Universal Robots PolyScope program: cognex01.urp

Program cognex01 (installation=default directory=/programs createdIn=5.9.1.1031110 lastSavedIn=5.9.1.1031110 robotSerialNumber=20195501059)
Calibrated DH parameters: a=[0.000146, -0.418764, -0.053981, 0.000058, -0.000023, 0]; d=[0.162545, 37.319448, -206.067439, 168.881546, 0.09955, 0.099464]; alpha=[1.57004, -0.001979, 0.002304, 1.570607, -1.57066, 0]; deltaTheta=[0, -0.174616, -1.258233, 1.432844, -0.000001, 0]
Robot Program (runOnlyOnce=false)
  URCap Cognex Camera Pose (Cognex In-Sight Robot Guidance, Cognex Corporation) dataModel(newNode=false, zLock=true, Variable(key=selectedVar, variable(name=CGX_result)))
    URCap Job Pass (Cognex In-Sight Robot Guidance, Cognex Corporation)
      MoveL speed 250 mm/s, acceleration 1200 mm/s^2 (useActiveTCP=true) feature=Base
        Waypoint Waypoint (Variable): variable=CGX_result
    URCap Job Fail (Cognex In-Sight Robot Guidance, Cognex Corporation)
      Placeholder
    URCap No Response (Cognex In-Sight Robot Guidance, Cognex Corporation)
      Placeholder
